PROGRAM Lectura_Maestro
VAR
	// >>>>>>>>>>>>>>>>>>>>>>>>>>>>>>>>>>>>>>>>   Estructuras de configuración con la comunicación desde y hacia el PLC Maestro <<<<<<<<<<<<<<<<<<<<<<<<<<<<<<<<<<<<<<<<<<<<<<<<<
	
	//Recordar que el IDXOFFS debe ser el doble de la posición a la que queréis acceder Ejemplo: para leer los strings a partir de la dirección MW100 Debéis poner 200 en exadecimal (C8)
	
//Configuración de la lectura de las variables Bool, IDXGRP:=16#4020(Hace referencia a la lectura de M),IDXOFFS:=16#B48C(Offset %MB46.220,  %MB46.220 a %MB46320), LEN : 101 Longitud bools leidos,DESTADDR:= ADR(Lectura_PLCs.aMasterBoolCom) Ubicación del array donde se guarda la lectura
	Config_Read_ADS_Bools_Maestro:Str_Config_ADS_to_PLC:=(NETID:='192.168.10.71.1.1', PORT:=851, IDXGRP:=16#4020,IDXOFFS:=16#B48C,LEN:=101,DESTADDR:= ADR(Lectura_PLCs.aMasterBoolCom));
	
	//Configuración de la lectura de las variables String, IDXGRP:=16#4020(Hace referencia a la lectura de M),IDXOFFS:= 16#14500(%MW42600 a %MW43815 ( 15 word)),Longitud de bytes a leer 1215 bytes = 15 strings que son 81words por cada string. ,DESTADDR:= ADR(Lectura_PLCs.aMasterStringCom) Ubicación del array donde se guarda la lectura
	Config_Read_ADS_Strings_Maestro:Str_Config_ADS_to_PLC:=(NETID:='192.168.10.71.1.1', PORT:=851, IDXGRP:=16#4020,IDXOFFS:=16#14500,LEN:=1215,DESTADDR:= ADR(Lectura_PLCs.aMasterStringCom));
	
	//Configuración de la lectura de las variables Times, IDXGRP:=16#4020(Hace referencia a la lectura de M),IDXOFFS:=16#17278 ( %MW47420 a %MW47614 (204 word),LEN:= 204 Longitud de bytes a leer bytes = 200words    51 componentes,DESTADDR:= ADR(Lectura_PLCs.aMasterTimeCom) Ubicación del array donde se guarda la lectura
	Config_Read_ADS_Times_Maestro:Str_Config_ADS_to_PLC:=(NETID:='192.168.10.71.1.1', PORT:=851, IDXGRP:=16#4020,IDXOFFS:=16#17278,LEN:= 204,DESTADDR:= ADR(Lectura_PLCs.aMasterTimeCom));
	
	//Configuración de la lectura de las variables Words, IDXGRP:=16#4020(Hace referencia a la lectura de M),IDXOFFS:=16#16008 ( %MW45060 a %MW45100 (40 word),82;//Longitud de bytes a leer 80 bytes = 40words   ,DESTADDR:= ADR(Lectura_PLCs.aMasteWordCom) Ubicación del array donde se guarda la lectura
	Config_Read_ADS_Words_Maestro:Str_Config_ADS_to_PLC:=(NETID:='192.168.10.71.1.1', PORT:=851, IDXGRP:=16#4020,IDXOFFS:=16#16008,LEN:=82,DESTADDR:= ADR(Lectura_PLCs.aMasterWordCom));
	
	fbLectura_a_PLC_Maestro:fbLectura_a_PLC;
	

END_VAR
VAR_INPUT
	bNextBlockToRead_L4_Done:BOOL;
END_VAR

fbLectura_a_PLC_Maestro(
	Config_PLC_ADS_Bools:=Config_Read_ADS_Bools_Maestro,
	Config_PLC_ADS_Strings:=Config_Read_ADS_Strings_Maestro,
	Config_PLC_ADS_Times:=Config_Read_ADS_Times_Maestro,
	Config_PLC_ADS_Words:=Config_Read_ADS_Words_Maestro,
 	TimeReadStateEntreLecturas:=T#20MS,
	bHabilitadaLectura:=TRUE,
	);

END_PROGRAM

(* stored: Version 1.1.0.1, ProductVersion 3.1.4024.12
   POU Lectura_Maestro: Id {61329b2f-9e3b-4ccf-999f-e1fad82321e2}, SpecialFunc None *)
